PROGRAM TestSimpleEstimatorANDController
VAR
	//inputs
	ErrorPose AT%I*: RobotPoseSimple;
	//Outputs
	nextWP AT%Q*: RobotPoseSimple;
	P, I, D, N AT%Q*: LREAL;
END_VAR

nextWP.x:=5150;
nextWP.y:=1560;
nextWP.theta:=0;
P:=1;
I:=0;
D:=0;
N:=100;

END_PROGRAM

(* stored: Version 1.1.0.1, ProductVersion 3.1.4024.11
   POU TestSimpleEstimatorANDController: Id {61c80a2a-3fb9-47a1-947b-5d5e0c0438c0}, SpecialFunc None *)
